INTERFACE IPistonHorizontal

METHOD MoveLeft : TcoCore.ITcoTaskStatus
END_METHOD

METHOD MoveRight : TcoCore.ITcoTaskStatus
END_METHOD

END_INTERFACE

(* stored: Version 1.1.0.1, ProductVersion 3.1.4024.9
   Itf IPistonHorizontal: Id {bbbdd7fb-23d4-0127-079c-3e0c6dc72306}
   Folder Horizontal: Id {2ff8d3b2-cc5c-0181-2275-d627c6d6b875}
   Method MoveLeft: Id {fd646f16-8520-0cfd-3cad-7317a6a08ccc}
   Method MoveRight: Id {3d107b04-8158-05bf-0a09-3ccb893cf2aa} *)
